{library PRIVATE}
(*
  Private Funtcion:
  Get the size for a datagram struct. The SIZEOF operator does not work on all systems. In all cases this function is safer.
*)
FUNCTION _DataGramSize : INT  
VAR_INPUT
END_VAR
VAR
	Data: 	DataGram;
END_VAR

 _DataGramSize:=SIZEOF(Data);
  
(* Enable this row if SIZEOF() does not work *)
(* _DataGramSize:=8; *)

END_FUNCTION

(* stored: Version 1.1.0.1, ProductVersion 3.1.4024.2
   POU _DataGramSize: Id {1d42ad0e-ac6e-4725-9472-a3e7f6836acd}, SpecialFunc None *)
